TYPE SxDuoCommand :
STRUCT
	ActivateFireAlarm: BOOL;
	ResetSmokeDetector: BOOL;
	ForceExercise: BOOL;	
END_STRUCT
END_TYPE

(* stored: Version 1.1.0.1, ProductVersion 3.1.4024.6
   DUT SxDuoCommand: Id {f3bc2133-a027-40ac-b4a0-5029b99faa89} *)
